// SIMATIC STEP 7 (V5.x) project ActuatorValve
// CPU: CPU 317F-2 PN/DP
// station: P_ADR_BUS
// station: Hardware
// station: SIMATIC 300(1)
// program: S7 Program(1)

SYMBOL_TABLE
"Valve01"	DB 1	FB 1
"ActuatorValceControl"	FB 1	FB 1
"ManualUp"	I 0.0	BOOL
"ManualDown"	I 0.1	BOOL
"Valve01Act"	IW 272	INT
"100ms"	M 0.0	BOOL
"200ms"	M 0.1	BOOL
"400ms"	M 0.2	BOOL
"500ms"	M 0.3	BOOL
"800ms"	M 0.4	BOOL
"1000ms"	M 0.5	BOOL
"1600ms"	M 0.6	BOOL
"2000ms"	M 0.7	BOOL
"100msMemory"	M 1.0	BOOL
"200msMemory"	M 1.1	BOOL
"400msMemory"	M 1.2	BOOL
"500msMemory"	M 1.3	BOOL
"800msMemory"	M 1.4	BOOL
"1000msMemory"	M 1.5	BOOL
"1600msMemory"	M 1.6	BOOL
"2000msMemory"	M 1.7	BOOL
"100msP_Edge"	M 2.0	BOOL
"200msP_Edge"	M 2.1	BOOL
"400msP_Edge"	M 2.2	BOOL
"500msP_Edge"	M 2.3	BOOL
"800msP_Edge"	M 2.4	BOOL
"1000msP_Edge"	M 2.5	BOOL
"1600msP_Edge"	M 2.6	BOOL
"2000msP_Edge"	M 2.7	BOOL
"AlwayTrue"	M 3.0	BOOL
"AlwayFalse"	M 3.1	BOOL
"EmptyTempoInt"	MW 100	WORD
"CYCL_EXC"	OB 1	OB 1	// Cycle Execution
"Valve01_Up"	Q 0.0	BOOL
"Valve01_Down"	Q 0.1	BOOL
"Valve01_Monitor"	VAT 1	
END_SYMBOL_TABLE

FUNCTION_BLOCK "ActuatorValceControl"	// FB 1
VERSION : 0.0
VAR_INPUT
  Tricker : BOOL ;	//INT := 7 ;
  PotenActual : INT ;
  ManualUp : BOOL ;
  ManualDown : BOOL ;
END_VAR
VAR_OUTPUT
  UpDirection : BOOL ;
  DownDirection : BOOL ;
END_VAR
VAR
  FullCyc : INT ;
  Start : BOOL ;
  UnderRunning : BOOL ;
  Stop : BOOL ;
  ClearActual : BOOL ;
  SetMin : BOOL ;
  SetMax : BOOL ;
  RunMode : INT ;
  OldRunMode : INT ;
  CycCounter : INT ;
  Up_Dir : BOOL ;
  Down_Dir : BOOL ;
  SwapDelay_Set : INT ;
  UpDelayAct : INT ;
  DownDelayAct : INT ;
  RecordDelay_Set : INT ;
  UpRecordAct : INT ;
  DownRecordAct : INT ;
  IndexUp : INT ;
  IndexDown : INT ;
  ActualTimeUp : INT ;
  ActualTimeDown : INT ;
  AutoMin : INT ;
  AutoMax : INT ;
  CalibrateUp : INT ;
  CalibrateDown : INT ;
  CalibrateLayer : INT ;
  DelayCalibrateSet : INT ;
  Del_Cal_Up_Act : INT ;
  Del_Cal_Down_Act : INT ;
  DelayCalCheckSet : INT ;	//Cross Check for Calibrate Function
  DelayCalCheckAct : INT ;	//Cross Check for Calibrate Function
  CalibrateError : BOOL ;
  PotenDistance : INT ;
  ManActPosiPercent : REAL ;
  ManualDistanceError : BOOL ;
  ManualLimitLowError : BOOL ;
  ManualLimitHiError : BOOL ;
  CalibrateSuccessfully : BOOL ;
  PotenSlip : INT ;
  PotenDistanceOK : INT ;
  ManualSetpoint : REAL ;
  ManualUpDirection : BOOL ;
  ManualDownDirection : BOOL ;
  ResetFaultManual : BOOL ;
  ManualSetOpposite : BOOL ;
  ManualSetAcceptGap : REAL ;
  ActualUp : ARRAY  [1 .. 100 ] OF INT ;
  ActualDown : ARRAY  [1 .. 100 ] OF INT ;
  TimeUp : ARRAY  [1 .. 100 ] OF INT ;
  TimeDown : ARRAY  [1 .. 100 ] OF INT ;
  DelayResetCalSet : INT ;
  DelayResetCalAct : INT ;
  ErrorCalAcceptance : INT ;
END_VAR
VAR_TEMP
  RealTemp01 : REAL ;
  IntTemp01 : INT ;
  I : INT ;
END_VAR
BEGIN
// body was compiled from an SCL source; compiled code not shown
END_FUNCTION_BLOCK

FUNCTION_BLOCK FB 2
VERSION : 0.0
VAR_INPUT
  Tricker : BOOL ;	//INT := 7 ;
  PotenActual : INT ;
  ManualUp : BOOL ;
  ManualDown : BOOL ;
END_VAR
VAR_OUTPUT
  UpDirection : BOOL ;
  DownDirection : BOOL ;
END_VAR
VAR
  FullCyc : INT ;
  Start : BOOL ;
  UnderRunning : BOOL ;
  Stop : BOOL ;
  ClearActual : BOOL ;
  SetMin : BOOL ;
  SetMax : BOOL ;
  RunMode : INT ;
  OldRunMode : INT ;
  CycCounter : INT ;
  Up_Dir : BOOL ;
  Down_Dir : BOOL ;
  SwapDelay_Set : INT ;
  UpDelayAct : INT ;
  DownDelayAct : INT ;
  RecordDelay_Set : INT ;
  UpRecordAct : INT ;
  DownRecordAct : INT ;
  IndexUp : INT ;
  IndexDown : INT ;
  ActualTimeUp : INT ;
  ActualTimeDown : INT ;
  AutoMin : INT ;
  AutoMax : INT ;
  CalibrateUp : INT ;
  CalibrateDown : INT ;
  CalibrateLayer : INT ;
  DelayCalibrateSet : INT ;
  Del_Cal_Up_Act : INT ;
  Del_Cal_Down_Act : INT ;
  DelayCalCheckSet : INT ;	//Cross Check for Calibrate Function
  DelayCalCheckAct : INT ;	//Cross Check for Calibrate Function
  CalibrateError : BOOL ;
  PotenDistance : INT ;
  ManActPosiPercent : REAL ;
  ManualDistanceError : BOOL ;
  ManualLimitLowError : BOOL ;
  ManualLimitHiError : BOOL ;
  CalibrateSuccessfully : BOOL ;
  PotenSlip : INT ;
  PotenDistanceOK : INT ;
  ManualSetpoint : REAL ;
  ManualUpDirection : BOOL ;
  ManualDownDirection : BOOL ;
  ResetFaultManual : BOOL ;
  ManualSetOpposite : BOOL ;
  ManualSetAcceptGap : REAL ;
  ActualUp : ARRAY  [1 .. 100 ] OF INT ;
  ActualDown : ARRAY  [1 .. 100 ] OF INT ;
  TimeUp : ARRAY  [1 .. 100 ] OF INT ;
  TimeDown : ARRAY  [1 .. 100 ] OF INT ;
  DelayResetCalSet : INT ;
  DelayResetCalAct : INT ;
  ErrorCalAcceptance : INT ;
END_VAR
VAR_TEMP
  RealTemp01 : REAL ;
  IntTemp01 : INT ;
  I : INT ;
END_VAR
BEGIN
// body was compiled from an SCL source; compiled code not shown
END_FUNCTION_BLOCK

DATA_BLOCK "Valve01"	// DB 1
VERSION : 0.0
"ActuatorValceControl"
BEGIN
END_DATA_BLOCK

ORGANIZATION_BLOCK "CYCL_EXC"	// OB 1
TITLE = "Main Program Sweep (Cycle)"
VERSION : 0.1
VAR_TEMP
  OB1_EV_CLASS : BYTE ;	//Bits 0-3 = 1 (Coming event), Bits 4-7 = 1 (Event class 1)
  OB1_SCAN_1 : BYTE ;	//1 (Cold restart scan 1 of OB 1), 3 (Scan 2-n of OB 1)
  OB1_PRIORITY : BYTE ;	//Priority of OB Execution
  OB1_OB_NUMBR : BYTE ;	//1 (Organization block 1, OB1)
  OB1_RESERVED_1 : BYTE ;	//Reserved for system
  OB1_RESERVED_2 : BYTE ;	//Reserved for system
  OB1_PREV_CYCLE : INT ;	//Cycle time of previous OB1 scan (milliseconds)
  OB1_MIN_CYCLE : INT ;	//Minimum cycle time of OB1 (milliseconds)
  OB1_MAX_CYCLE : INT ;	//Maximum cycle time of OB1 (milliseconds)
  OB1_DATE_TIME : DATE_AND_TIME ;	//Date and time OB1 started
END_VAR
BEGIN
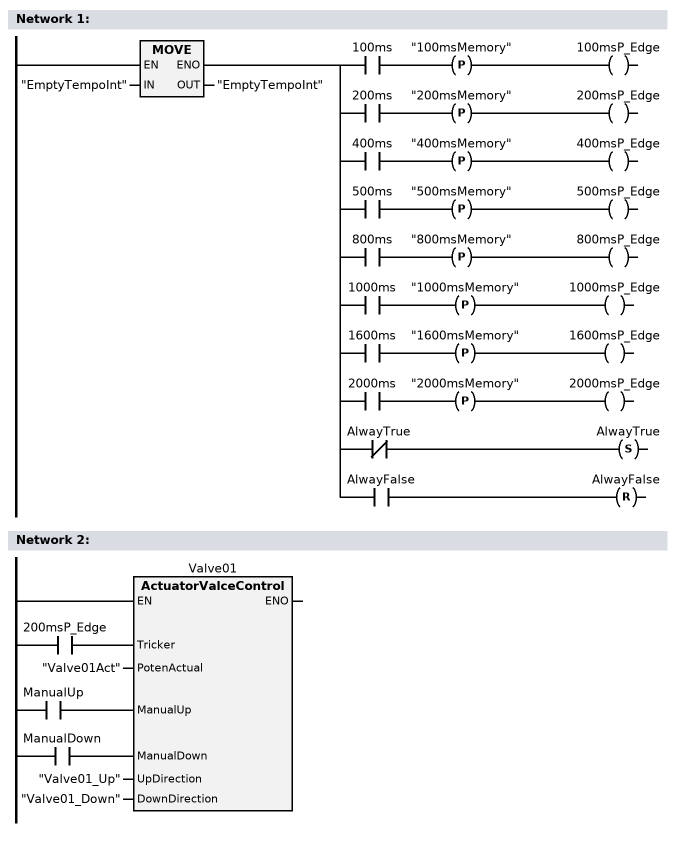
NETWORK
TITLE =
      L     "EmptyTempoInt";
      T     "EmptyTempoInt";
      SET;
      SAVE;
      CLR;
      A     BR;
      =     L 20.0;
      A     L 20.0;
      A     "100ms";
      FP    "100msMemory";
      =     "100msP_Edge";
      A     L 20.0;
      A     "200ms";
      FP    "200msMemory";
      =     "200msP_Edge";
      A     L 20.0;
      A     "400ms";
      FP    "400msMemory";
      =     "400msP_Edge";
      A     L 20.0;
      A     "500ms";
      FP    "500msMemory";
      =     "500msP_Edge";
      A     L 20.0;
      A     "800ms";
      FP    "800msMemory";
      =     "800msP_Edge";
      A     L 20.0;
      A     "1000ms";
      FP    "1000msMemory";
      =     "1000msP_Edge";
      A     L 20.0;
      A     "1600ms";
      FP    "1600msMemory";
      =     "1600msP_Edge";
      A     L 20.0;
      A     "2000ms";
      FP    "2000msMemory";
      =     "2000msP_Edge";
      A     L 20.0;
      AN    "AlwayTrue";
      S     "AlwayTrue";
      A     L 20.0;
      A     "AlwayFalse";
      R     "AlwayFalse";
NETWORK
TITLE =
      A     "200msP_Edge";
      =     L 20.0;
      BLD   103;
      A     "ManualUp";
      =     L 20.1;
      BLD   103;
      A     "ManualDown";
      =     L 20.2;
      BLD   103;
      CALL  "ActuatorValceControl" , "Valve01" (
           Tricker                  := L 20.0,
           PotenActual              := "Valve01Act",
           ManualUp                 := L 20.1,
           ManualDown               := L 20.2,
           UpDirection              := "Valve01_Up",
           DownDirection            := "Valve01_Down");
      NOP   0;
NETWORK
TITLE =
END_ORGANIZATION_BLOCK
